// TIA Portal project "Lab3" (V15)

(* hardware
DEVICE "S71500/ET200MP station_1"  S7-1500 station
   slot 0: "Rail_0"  Rack  6ES7 590-1***0-0AA0
   slot 1: "PLC_1"  CPU 1511-1 PN  6ES7 511-1AK00-0AB0  V1.0
      slot 3: "CPU display_1"  6ES7591-1XA00-0AA0
   slot 2: "DI 16x24VDC HF_1"  DI 16x24VDC HF  6ES7 521-1BH00-0AB0  V1.0
   slot 3: "DQ 16x24VDC/0.5A ST_1"  DQ 16x24VDC/0.5A ST  6ES7 522-1BH00-0AB0  V1.0
   slot 4: "AI 8xU/I/RTD/TC ST_1"  AI 8xU/I/RTD/TC ST  6ES7 531-7KF00-0AB0  V2.0
*)

// ===== PLC "PLC_1"  CPU 1511-1 PN =====

VAR_GLOBAL   // PLC tag table "Default tag table"
   "K1_L" AT %I0.0 : Bool;
   "K1_R" AT %I0.1 : Bool;
   "K2_L" AT %I0.2 : Bool;
   "K2_R" AT %I0.3 : Bool;
   "K3_L" AT %I0.4 : Bool;
   "K3_R" AT %I0.5 : Bool;
   "K4_L" AT %I0.6 : Bool;
   "K4_R" AT %I0.7 : Bool;
   "K1_CL" AT %Q0.0 : Bool;
   "K1_CR" AT %Q0.1 : Bool;
   "K2_CL" AT %Q0.2 : Bool;
   "K2_CR" AT %Q0.3 : Bool;
   "K3_CL" AT %Q0.4 : Bool;
   "K4_CL" AT %Q0.6 : Bool;
   "K1_P" AT %IW2 : Word;
   "K3_P" AT %IW4 : Word;
   "Cnt1" AT %C0 : Counter;
   "Cnt2" AT %C1 : Counter;
END_VAR

DATA_BLOCK "Lab2_DB"   // DB1
{ S7_Optimized_Access := 'TRUE' }
VERSION : 0.1
   VAR
      Done1 : Bool;
      Done2 : Bool;
      Done3 : Bool;
      Done4 : Bool;
      DoneWait : Bool;
      Set_Point_1 : Int;
      Set_Point_2 : Int;
      Set_Point_3 : Int;
      Set_Point_4 : Int;
      Reset : Bool;
      Discard1 : Bool;
      Discard2 : Bool;
   END_VAR
BEGIN
END_DATA_BLOCK

DATA_BLOCK "GRAFCET_DB"   // DB3
{ S7_Optimized_Access := 'TRUE' }
VERSION : 0.1
// stored: InstanceOfName GRAFCET
"GRAFCET"
BEGIN
END_DATA_BLOCK

FUNCTION_BLOCK "GRAFCET"   // FB2, GRAPH_PLUS
{ S7_Optimized_Access := 'TRUE' }
VERSION : 0.1
   VAR_INPUT
      OFF_SQ : Bool := false;   // Turn sequence off
      INIT_SQ : Bool := false;   // Set sequence to initial state
      ACK_EF : Bool := false;   // Acknowledge all errors and faults
      S_PREV : Bool := false;   // Output previous step in parameter S_NO
      S_NEXT : Bool := false;   // Indicate next step in parameter S_NO
      SW_AUTO : Bool := false;   // Automatic mode
      SW_TAP : Bool := false;   // Semiautomatic/switch with transition
      SW_TOP : Bool := false;   // Semiautomatic/ignore transition
      SW_MAN : Bool := false;   // Manual mode
      S_SEL : Int := 0;   // Select step to be output to S_NO
      S_ON : Bool := false;   // Activate step indicated in S_NO
      S_OFF : Bool := false;   // Deactivate step indicated S_NO
      T_PUSH : Bool := false;   // Enable transition to switch in semi automatic mode
   END_VAR
   VAR_OUTPUT
      S_NO : Int := 0;   // Step number
      S_MORE : Bool := false;   // More steps are available and can be shown in S_NO
      S_ACTIVE : Bool := false;   // Step indicated in S_NO is active
      ERR_FLT : Bool := false;   // Interlock or supervision group error
      AUTO_ON : Bool := false;   // Automatic mode is active
      TAP_ON : Bool := false;   // Semiautomatic mode/step with transition enabled
      TOP_ON : Bool := false;   // Semiautomatic mode/ignore transition enabled
      MAN_ON : Bool := false;   // Manual mode is active
   END_VAR
   VAR
      HMI_INFO : Array[0..8] of UInt;
      IF_PAR : G7_IfParPlus_V2;
      RT_DATA : G7_RTDataPlus_V2;   // Internal data area
      Trans1 : G7_TransitionPlus_V2;   // Transition structure
      Trans3 : G7_TransitionPlus_V2;   // Transition structure
      Trans4 : G7_TransitionPlus_V2;   // Transition structure
      Trans5 : G7_TransitionPlus_V2;   // Transition structure
      Trans6 : G7_TransitionPlus_V2;   // Transition structure
      Trans7 : G7_TransitionPlus_V2;   // Transition structure
      Trans8 : G7_TransitionPlus_V2;   // Transition structure
      Trans9 : G7_TransitionPlus_V2;   // Transition structure
      Trans10 : G7_TransitionPlus_V2;   // Transition structure
      Trans11 : G7_TransitionPlus_V2;   // Transition structure
      Trans12 : G7_TransitionPlus_V2;   // Transition structure
      Trans13 : G7_TransitionPlus_V2;   // Transition structure
      Trans14 : G7_TransitionPlus_V2;   // Transition structure
      Trans15 : G7_TransitionPlus_V2;   // Transition structure
      Trans16 : G7_TransitionPlus_V2;   // Transition structure
      Prazno : G7_StepPlus_V2;   // Step structure
      Inicijalizacija : G7_StepPlus_V2;   // Step structure
      "K2 levo" : G7_StepPlus_V2;   // Step structure
      "K4 levo" : G7_StepPlus_V2;   // Step structure
      "K1 50%" : G7_StepPlus_V2;   // Step structure
      "K3 levo" : G7_StepPlus_V2;   // Step structure
      "K1 desno" : G7_StepPlus_V2;   // Step structure
      "K3 75%" : G7_StepPlus_V2;   // Step structure
      "K2 desno" : G7_StepPlus_V2;   // Step structure
      "Cekaj 10s" : G7_StepPlus_V2;   // Step structure
      "K3 desno" : G7_StepPlus_V2;   // Step structure
      "K4 desno" : G7_StepPlus_V2;   // Step structure
      Resetovanje : G7_StepPlus_V2;   // Step structure
      SINI : Array[0..1] of USInt;
      LSTT : Array[0..14] of USInt;
      ATAJ : Array[0..14] of USInt;
      ATAB : Array[0..14] of USInt;
      PSTT : Array[0..14] of USInt;
      NSTT : Array[0..14] of USInt;
      ASSJ : Array[0..12] of USInt;
      ASSB : Array[0..12] of USInt;
      PTTS : Array[0..12] of USInt;
      NTTS : Array[0..12] of USInt;
      SW_SQTS : Array[0..12] of USInt;
      SWITCH : Array[0..1] of USInt;
      TVX : Array[0..5] of USInt;
      TTX : Array[0..5] of USInt;
      TSX : Array[0..1] of USInt;
      S00X : Array[0..1] of USInt;
      SOFFX : Array[0..1] of USInt;
      SONX : Array[0..1] of USInt;
      SAX : Array[0..1] of USInt;
      SERRX : Array[0..13] of USInt;
      SMX : Array[0..13] of USInt;
      S0X : Array[0..13] of USInt;
      S1X : Array[0..13] of USInt;
      IL_ALARM_INST : Program_Alarm;
      SUP_ALARM_INST : Program_Alarm;
      STEP_TIME_ALARM_INST : Program_Alarm;
      IEC_TIMER_INST : IEC_TIMER;
      TRANSACTION_FLAG : Bool := false;
   END_VAR
   // SINI[0] := 2;
   // LSTT[0] := 255;
   // LSTT[1] := 255;
   // LSTT[2] := 255;
   // LSTT[3] := 255;
   // LSTT[4] := 255;
   // LSTT[5] := 255;
   // LSTT[6] := 255;
   // LSTT[7] := 255;
   // LSTT[8] := 255;
   // LSTT[9] := 255;
   // LSTT[10] := 255;
   // LSTT[11] := 4;
   // LSTT[12] := 2;
   // LSTT[13] := 255;
   // ATAJ[1] := 1;
   // ATAJ[2] := 2;
   // ATAJ[3] := 3;
   // ATAJ[4] := 4;
   // ATAJ[5] := 5;
   // ATAJ[6] := 6;
   // ATAJ[7] := 7;
   // ATAJ[8] := 8;
   // ATAJ[9] := 9;
   // ATAJ[10] := 10;
   // ATAJ[11] := 11;
   // ATAJ[12] := 12;
   // ATAJ[13] := 13;
   // ATAB[1] := 1;
   // ATAB[2] := 2;
   // ATAB[3] := 3;
   // ATAB[4] := 4;
   // ATAB[5] := 5;
   // ATAB[6] := 11;
   // ATAB[7] := 7;
   // ATAB[8] := 8;
   // ATAB[9] := 9;
   // ATAB[10] := 12;
   // ATAB[11] := 6;
   // ATAB[12] := 10;
   // ATAB[13] := 13;
   // PSTT[1] := 2;
   // PSTT[2] := 3;
   // PSTT[3] := 4;
   // PSTT[4] := 5;
   // PSTT[5] := 6;
   // PSTT[6] := 7;
   // PSTT[7] := 8;
   // PSTT[8] := 9;
   // PSTT[9] := 10;
   // PSTT[10] := 11;
   // PSTT[11] := 7;
   // PSTT[12] := 11;
   // PSTT[13] := 1;
   // NSTT[0] := 1;
   // NSTT[1] := 3;
   // NSTT[2] := 4;
   // NSTT[3] := 5;
   // NSTT[4] := 6;
   // NSTT[5] := 7;
   // NSTT[6] := 8;
   // NSTT[7] := 9;
   // NSTT[8] := 10;
   // NSTT[9] := 11;
   // NSTT[10] := 12;
   // NSTT[11] := 4;
   // NSTT[12] := 2;
   // NSTT[13] := 2;
   // ASSJ[1] := 1;
   // ASSJ[2] := 2;
   // ASSJ[3] := 3;
   // ASSJ[4] := 4;
   // ASSJ[5] := 5;
   // ASSJ[6] := 6;
   // ASSJ[7] := 7;
   // ASSJ[8] := 8;
   // ASSJ[9] := 9;
   // ASSJ[10] := 10;
   // ASSJ[11] := 11;
   // ASSB[1] := 1;
   // ASSB[2] := 2;
   // ASSB[3] := 3;
   // ASSB[4] := 4;
   // ASSB[5] := 5;
   // ASSB[6] := 6;
   // ASSB[7] := 7;
   // ASSB[8] := 8;
   // ASSB[9] := 9;
   // ASSB[10] := 10;
   // ASSB[11] := 11;
   // PTTS[0] := 255;
   // PTTS[2] := 13;
   // PTTS[3] := 1;
   // PTTS[4] := 2;
   // PTTS[5] := 3;
   // PTTS[6] := 4;
   // PTTS[7] := 5;
   // PTTS[8] := 6;
   // PTTS[9] := 7;
   // PTTS[10] := 8;
   // PTTS[11] := 9;
   // NTTS[1] := 13;
   // NTTS[2] := 1;
   // NTTS[3] := 2;
   // NTTS[4] := 3;
   // NTTS[5] := 4;
   // NTTS[6] := 5;
   // NTTS[7] := 6;
   // NTTS[8] := 7;
   // NTTS[9] := 8;
   // NTTS[10] := 9;
   // NTTS[11] := 10;
   // SW_SQTS[8] := 1;
   // SW_SQTS[9] := 1;
   // SW_SQTS[10] := 1;
   // SW_SQTS[11] := 1;
   // TVX[0] := 16#1;
   // TTX[0] := 16#1;
   // TSX[0] := 16#1;
   // S00X[0] := 16#1;
   // SOFFX[0] := 16#1;
   // SONX[0] := 16#1;
   // SAX[0] := 16#1;
   // SERRX[0] := 16#1;
   // SMX[0] := 16#1;
   // S0X[0] := 16#1;
   // S1X[0] := 16#1;
   // LSTT[14] := 1;
   // ATAJ[14] := 14;
   // ATAB[14] := 14;
   // PSTT[14] := 12;
   // NSTT[14] := 1;
   // ASSJ[12] := 12;
   // ASSB[12] := 12;
   // PTTS[12] := 10;
   // NTTS[12] := 14;
   // SW_SQTS[12] := 2;
BEGIN
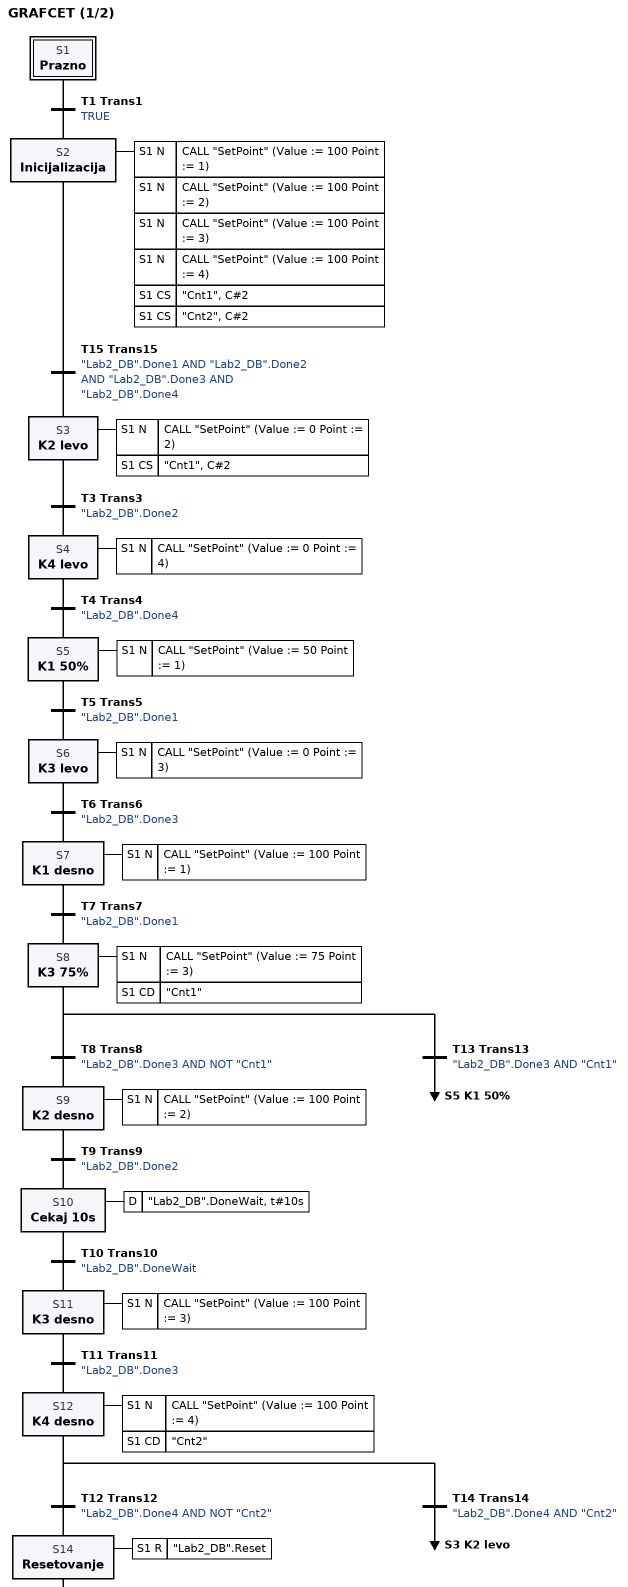
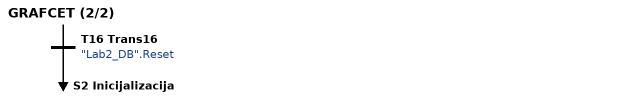
   // sequencer 1
   INITIAL_STEP Prazno:   // S1, max time T#10S, warning time T#7S
   END_STEP
   TRANSITION Trans1 FROM Prazno TO Inicijalizacija   // T1
      := TRUE;
   END_TRANSITION
   STEP Inicijalizacija:   // S2, max time T#10S, warning time T#7S
          S1  N    CALL "SetPoint" (Value := 100 Point := 1)
          S1  N    CALL "SetPoint" (Value := 100 Point := 2)
          S1  N    CALL "SetPoint" (Value := 100 Point := 3)
          S1  N    CALL "SetPoint" (Value := 100 Point := 4)
          S1  CS   "Cnt1", C#2
          S1  CS   "Cnt2", C#2
   END_STEP
   TRANSITION Trans15 FROM Inicijalizacija TO "K2 levo"   // T15
      := "Lab2_DB".Done1 AND "Lab2_DB".Done2 AND "Lab2_DB".Done3 AND "Lab2_DB".Done4;
   END_TRANSITION
   STEP "K2 levo":   // S3, max time T#10S, warning time T#7S
          S1  N    CALL "SetPoint" (Value := 0 Point := 2)
          S1  CS   "Cnt1", C#2
   END_STEP
   TRANSITION Trans3 FROM "K2 levo" TO "K4 levo"   // T3
      := "Lab2_DB".Done2;
   END_TRANSITION
   STEP "K4 levo":   // S4, max time T#10S, warning time T#7S
          S1  N    CALL "SetPoint" (Value := 0 Point := 4)
   END_STEP
   TRANSITION Trans4 FROM "K4 levo" TO "K1 50%"   // T4
      := "Lab2_DB".Done4;
   END_TRANSITION
   STEP "K1 50%":   // S5, max time T#10S, warning time T#7S
          S1  N    CALL "SetPoint" (Value := 50 Point := 1)
   END_STEP
   TRANSITION Trans5 FROM "K1 50%" TO "K3 levo"   // T5
      := "Lab2_DB".Done1;
   END_TRANSITION
   STEP "K3 levo":   // S6, max time T#10S, warning time T#7S
          S1  N    CALL "SetPoint" (Value := 0 Point := 3)
   END_STEP
   TRANSITION Trans6 FROM "K3 levo" TO "K1 desno"   // T6
      := "Lab2_DB".Done3;
   END_TRANSITION
   STEP "K1 desno":   // S7, max time T#10S, warning time T#7S
          S1  N    CALL "SetPoint" (Value := 100 Point := 1)
   END_STEP
   TRANSITION Trans7 FROM "K1 desno" TO "K3 75%"   // T7
      := "Lab2_DB".Done1;
   END_TRANSITION
   STEP "K3 75%":   // S8, max time T#10S, warning time T#7S
          S1  N    CALL "SetPoint" (Value := 75 Point := 3)
          S1  CD   "Cnt1"
   END_STEP
   TRANSITION Trans8 FROM "K3 75%" TO "K2 desno"   // T8
      := "Lab2_DB".Done3 AND NOT "Cnt1";
   END_TRANSITION
   TRANSITION Trans13 FROM "K3 75%" TO "K1 50%"   // T13, jump
      := "Lab2_DB".Done3 AND "Cnt1";
   END_TRANSITION
   STEP "K2 desno":   // S9, max time T#10S, warning time T#7S
          S1  N    CALL "SetPoint" (Value := 100 Point := 2)
   END_STEP
   TRANSITION Trans9 FROM "K2 desno" TO "Cekaj 10s"   // T9
      := "Lab2_DB".Done2;
   END_TRANSITION
   STEP "Cekaj 10s":   // S10, max time T#10S, warning time T#7S
              D    "Lab2_DB".DoneWait, t#10s
   END_STEP
   TRANSITION Trans10 FROM "Cekaj 10s" TO "K3 desno"   // T10
      := "Lab2_DB".DoneWait;
   END_TRANSITION
   STEP "K3 desno":   // S11, max time T#10S, warning time T#7S
          S1  N    CALL "SetPoint" (Value := 100 Point := 3)
   END_STEP
   TRANSITION Trans11 FROM "K3 desno" TO "K4 desno"   // T11
      := "Lab2_DB".Done3;
   END_TRANSITION
   STEP "K4 desno":   // S12, max time T#10S, warning time T#7S
          S1  N    CALL "SetPoint" (Value := 100 Point := 4)
          S1  CD   "Cnt2"
   END_STEP
   TRANSITION Trans12 FROM "K4 desno" TO Resetovanje   // T12
      := "Lab2_DB".Done4 AND NOT "Cnt2";
   END_TRANSITION
   TRANSITION Trans14 FROM "K4 desno" TO "K2 levo"   // T14, jump
      := "Lab2_DB".Done4 AND "Cnt2";
   END_TRANSITION
   STEP Resetovanje:   // S14, max time T#10S, warning time T#7S
          S1  R    "Lab2_DB".Reset
   END_STEP
   TRANSITION Trans16 FROM Resetovanje TO Inicijalizacija   // T16, jump
      := "Lab2_DB".Reset;
   END_TRANSITION
END_FUNCTION_BLOCK

FUNCTION "SetPoint" : Void   // FC1, LAD
{ S7_Optimized_Access := 'TRUE' }
VERSION : 0.1
   VAR_INPUT
      Value : Int;
      Point : Int;
   END_VAR
BEGIN

REGION Network 1
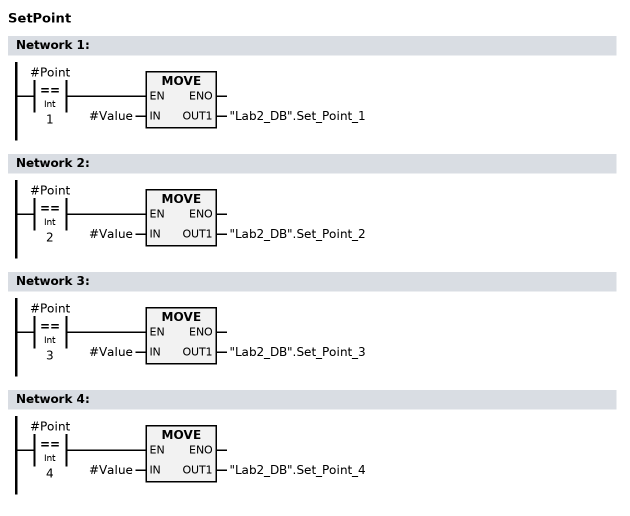
   RUNG wire#powerrail
      { S7_Templates := "SrcType := Int" } EQ_Contact(in1 := #Point, in2 := 1)
      Move(in := #Value, out1 => "Lab2_DB".Set_Point_1)
   END_RUNG
   // the same network as SCL:
   IF #Point = 1 THEN "Lab2_DB".Set_Point_1 := #Value; END_IF;
END_REGION

REGION Network 2
   RUNG wire#powerrail
      { S7_Templates := "SrcType := Int" } EQ_Contact(in1 := #Point, in2 := 2)
      Move(in := #Value, out1 => "Lab2_DB".Set_Point_2)
   END_RUNG
   // the same network as SCL:
   IF #Point = 2 THEN "Lab2_DB".Set_Point_2 := #Value; END_IF;
END_REGION

REGION Network 3
   RUNG wire#powerrail
      { S7_Templates := "SrcType := Int" } EQ_Contact(in1 := #Point, in2 := 3)
      Move(in := #Value, out1 => "Lab2_DB".Set_Point_3)
   END_RUNG
   // the same network as SCL:
   IF #Point = 3 THEN "Lab2_DB".Set_Point_3 := #Value; END_IF;
END_REGION

REGION Network 4
   RUNG wire#powerrail
      { S7_Templates := "SrcType := Int" } EQ_Contact(in1 := #Point, in2 := 4)
      Move(in := #Value, out1 => "Lab2_DB".Set_Point_4)
   END_RUNG
   // the same network as SCL:
   IF #Point = 4 THEN "Lab2_DB".Set_Point_4 := #Value; END_IF;
END_REGION
END_FUNCTION

FUNCTION "Lab2_Motion_Control" : Void   // FC3, LAD
{ S7_Optimized_Access := 'TRUE' }
VERSION : 0.1
   VAR_INPUT
      Set_Point : Int;
      Sensor_Left : Bool;
      Sensor_Right : Bool;
      Sensor_Analog : Int;
   END_VAR
   VAR_OUTPUT
      Move_Left : Bool;
      Move_Right : Bool;
      Done : Bool;
   END_VAR
   VAR_TEMP
      Target_Value : Int;
      Current_Value : Int;
      Tmp_Diff : Int;
      Tmp_ADiff : Int;
   END_VAR
   VAR_TEMP   // added for the SCL form of the ladder/FBD networks
      _w1 : Bool;
   END_VAR
BEGIN

REGION Network 1
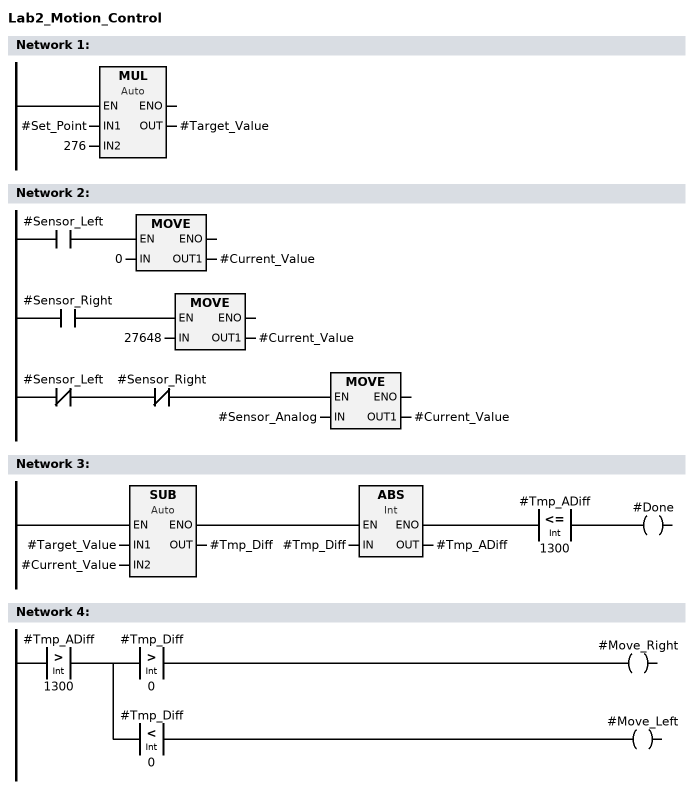
   RUNG wire#powerrail
      Mul(in1 := #Set_Point, in2 := 276, out => #Target_Value)
   END_RUNG
   // the same network as SCL:
   #Target_Value := #Set_Point * 276;
END_REGION

REGION Network 2
   RUNG wire#powerrail
      Contact( #Sensor_Left )
      Move(in := 0, out1 => #Current_Value)
   END_RUNG
   RUNG wire#powerrail
      Contact( #Sensor_Right )
      Move(in := 27648, out1 => #Current_Value)
   END_RUNG
   RUNG wire#powerrail
      I_Contact( #Sensor_Left )
      I_Contact( #Sensor_Right )
      Move(in := #Sensor_Analog, out1 => #Current_Value)
   END_RUNG
   // the same network as SCL:
   IF #Sensor_Left THEN #Current_Value := 0; END_IF;
   IF #Sensor_Right THEN #Current_Value := 27648; END_IF;
   IF NOT #Sensor_Left AND NOT #Sensor_Right THEN #Current_Value := #Sensor_Analog; END_IF;
END_REGION

REGION Network 3
   RUNG wire#powerrail
      Sub(in1 := #Target_Value, in2 := #Current_Value, out => #Tmp_Diff)
      { S7_Templates := "SrcType := Int" } Abs(in := #Tmp_Diff, out => #Tmp_ADiff)
      { S7_Templates := "SrcType := Int" } LE_Contact(in1 := #Tmp_ADiff, in2 := 1300)
      Coil( #Done )
   END_RUNG
   // the same network as SCL:
   #Tmp_Diff := #Target_Value - #Current_Value;
   #Tmp_ADiff := ABS(#Tmp_Diff);
   #Done := #Tmp_ADiff <= 1300;
END_REGION

REGION Network 4
   RUNG wire#powerrail
      { S7_Templates := "SrcType := Int" } GT_Contact(in1 := #Tmp_ADiff, in2 := 1300)
      wire#w1
      { S7_Templates := "SrcType := Int" } GT_Contact(in1 := #Tmp_Diff, in2 := 0)
      Coil( #Move_Right )
   END_RUNG
   RUNG wire#w1
      { S7_Templates := "SrcType := Int" } LT_Contact(in1 := #Tmp_Diff, in2 := 0)
      Coil( #Move_Left )
   END_RUNG
   // the same network as SCL:
   #_w1 := #Tmp_ADiff > 1300;
   #Move_Right := #_w1 AND (#Tmp_Diff > 0);
   #Move_Left := #_w1 AND (#Tmp_Diff < 0);
END_REGION
END_FUNCTION

ORGANIZATION_BLOCK "Main"   // OB1, LAD, ProgramCycle
TITLE = "Main Program Sweep (Cycle)"
{ S7_Optimized_Access := 'TRUE' }
VERSION : 0.1
   VAR_INPUT
      Initial_Call : Bool;   // Initial call of this OB
      Remanence : Bool;   // =True, if remanent data are available
   END_VAR
   VAR_TEMP   // added for the SCL form of the ladder/FBD networks
      _w1 : Bool;
      _w2 : Bool;
      _w3 : Bool;
   END_VAR
BEGIN

REGION Network 1
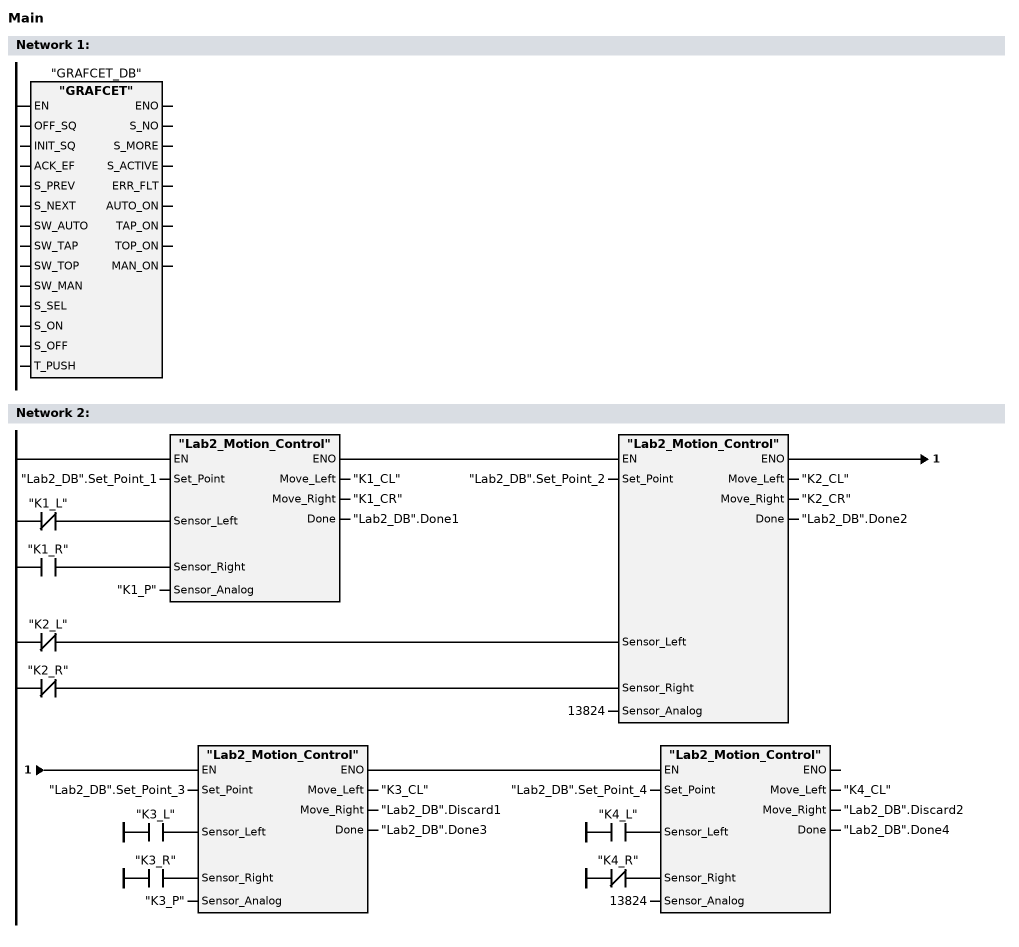
   RUNG wire#powerrail
      "GRAFCET_DB"(OFF_SQ :=, INIT_SQ :=, ACK_EF :=, S_PREV :=, S_NEXT :=, SW_AUTO :=, SW_TAP :=, SW_TOP :=, SW_MAN :=, S_SEL :=, S_ON :=, S_OFF :=, T_PUSH :=, S_NO =>, S_MORE =>, S_ACTIVE =>, ERR_FLT =>, AUTO_ON =>, TAP_ON =>, TOP_ON =>, MAN_ON =>)
   END_RUNG
   // the same network as SCL:
   "GRAFCET_DB"();   // "GRAFCET"
END_REGION

REGION Network 2
   RUNG wire#powerrail
      "Lab2_Motion_Control"(Sensor_Left := wire#w1, Sensor_Right := wire#w2, Set_Point := "Lab2_DB".Set_Point_1, Sensor_Analog := "K1_P", Move_Left => "K1_CL", Move_Right => "K1_CR", Done => "Lab2_DB".Done1)
      "Lab2_Motion_Control"(Sensor_Left := wire#w3, Sensor_Right := wire#w4, Set_Point := "Lab2_DB".Set_Point_2, Sensor_Analog := 13824, Move_Left => "K2_CL", Move_Right => "K2_CR", Done => "Lab2_DB".Done2)
      "Lab2_Motion_Control"(Sensor_Left := wire#w5, Sensor_Right := wire#w6, Set_Point := "Lab2_DB".Set_Point_3, Sensor_Analog := "K3_P", Move_Left => "K3_CL", Move_Right => "Lab2_DB".Discard1, Done => "Lab2_DB".Done3)
      "Lab2_Motion_Control"(Sensor_Left := wire#w7, Sensor_Right := wire#w8, Set_Point := "Lab2_DB".Set_Point_4, Sensor_Analog := 13824, Move_Left => "K4_CL", Move_Right => "Lab2_DB".Discard2, Done => "Lab2_DB".Done4)
   END_RUNG
   RUNG wire#powerrail
      I_Contact( "K1_L" )
   END_RUNG wire#w1
   RUNG wire#powerrail
      Contact( "K1_R" )
   END_RUNG wire#w2
   RUNG wire#powerrail
      I_Contact( "K2_L" )
   END_RUNG wire#w3
   RUNG wire#powerrail
      I_Contact( "K2_R" )
   END_RUNG wire#w4
   RUNG wire#powerrail
      Contact( "K3_L" )
   END_RUNG wire#w5
   RUNG wire#powerrail
      Contact( "K3_R" )
   END_RUNG wire#w6
   RUNG wire#powerrail
      Contact( "K4_L" )
   END_RUNG wire#w7
   RUNG wire#powerrail
      I_Contact( "K4_R" )
   END_RUNG wire#w8
   // the same network as SCL:
   "Lab2_Motion_Control"(Set_Point := "Lab2_DB".Set_Point_1,
                         Sensor_Left := NOT "K1_L",
                         Sensor_Right := "K1_R",
                         Sensor_Analog := "K1_P",
                         Move_Left => "K1_CL",
                         Move_Right => "K1_CR",
                         Done => "Lab2_DB".Done1,
                         ENO => #_w1);
   "Lab2_Motion_Control"(EN := #_w1,
                         Set_Point := "Lab2_DB".Set_Point_2,
                         Sensor_Left := NOT "K2_L",
                         Sensor_Right := NOT "K2_R",
                         Sensor_Analog := 13824,
                         Move_Left => "K2_CL",
                         Move_Right => "K2_CR",
                         Done => "Lab2_DB".Done2,
                         ENO => #_w2);
   "Lab2_Motion_Control"(EN := #_w2,
                         Set_Point := "Lab2_DB".Set_Point_3,
                         Sensor_Left := "K3_L",
                         Sensor_Right := "K3_R",
                         Sensor_Analog := "K3_P",
                         Move_Left => "K3_CL",
                         Move_Right => "Lab2_DB".Discard1,
                         Done => "Lab2_DB".Done3,
                         ENO => #_w3);
   IF #_w3 THEN
       "Lab2_Motion_Control"(Set_Point := "Lab2_DB".Set_Point_4,
                             Sensor_Left := "K4_L",
                             Sensor_Right := NOT "K4_R",
                             Sensor_Analog := 13824,
                             Move_Left => "K4_CL",
                             Move_Right => "Lab2_DB".Discard2,
                             Done => "Lab2_DB".Done4);
   END_IF;
END_REGION
END_ORGANIZATION_BLOCK